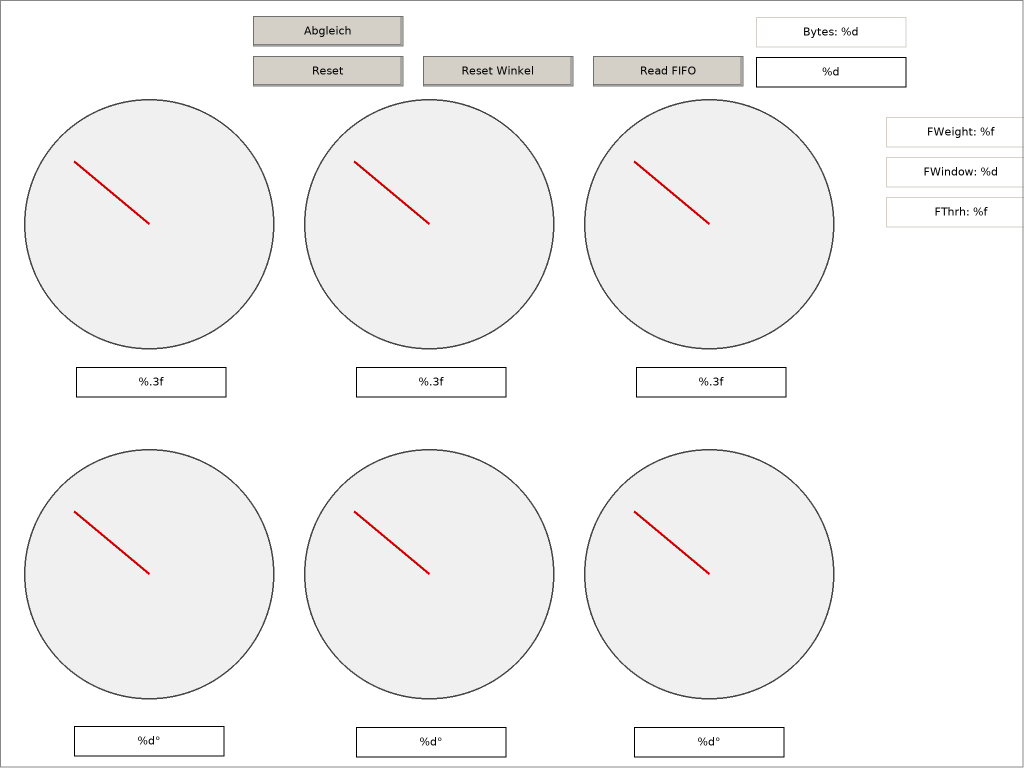
VISUALIZATION Visualization  // 1024x768
    Meter360 (24,99 250x250), value: MAIN.DegMovingHead[2], style: Meter-Meter360-Gray, scale format: %d, scale 0..360
    Rectangle (76,367 150x30), "%.3f", text variable: MAIN.Deg[0]
    Button (253,16 150x30), "Abgleich", colour toggle: MAIN.iFilter[0].bRingbufferFilled
        p2175578022: 16#ffffff
        p573394764: 16#FFFF8080
        tap MAIN.bWriteOffset
    Button (253,56 150x30), "Reset"
        tap MAIN.bReset
    Meter360 (304,99 250x250), value: MAIN.DegMovingHead[1], style: Meter-Meter360-Gray, scale format: %d, scale 0..360
    Rectangle (356,367 150x30), "%.3f", text variable: MAIN.Deg[1]
    Meter360 (584,99 250x250), value: MAIN.DegMovingHead[0], style: Meter-Meter360-Gray, scale format: %d, scale 0..360
    Rectangle (636,367 150x30), "%.3f", text variable: MAIN.Deg[0]
    Button (423,56 150x30), "Reset Winkel"
        tap MAIN.bResetAngle
    Button (593,56 150x30), "Read FIFO"
        tap MAIN.bReadFIFO
    Rectangle (756,57 150x30), "%d", text variable: MAIN.arBuf[2]
    Textfield (756,17 150x30), "Bytes: %d", text variable: MAIN.bytesToRead
        OnMouseClick: write the text variable via Default
    Meter360 (24,449 250x250), value: MAIN.degGamma, style: Meter-Meter360-Gray, scale format: %d, scale 0..360
    Meter360 (304,449 250x250), value: MAIN.degTheta, style: Meter-Meter360-Gray, scale format: %d, scale 0..360
    Meter360 (584,449 250x250), value: MAIN.degPhi, style: Meter-Meter360-Gray, scale format: %d, scale 0..360
    Textfield (886,117 150x30), "FWeight: %f", text variable: MAIN.fusionWeight
        OnMouseClick: write the text variable via Default
    Textfield (886,157 150x30), "FWindow: %d", text variable: MAIN.fusionWindow
        OnMouseClick: write the text variable via Default
    Textfield (886,197 150x30), "FThrh: %f", text variable: MAIN.fusionHorizontThreshold
        OnMouseClick: write the text variable via Default
    Rectangle (74,726 150x30), "%d°", text variable: MAIN.degGamma
    Rectangle (356,727 150x30), "%d°", text variable: MAIN.degTheta
    Rectangle (634,727 150x30), "%d°", text variable: MAIN.degTheta
END_VISUALIZATION

(* stored: Version 1.1.0.1, ProductVersion 3.1.4024.12
   Visu Visualization: Id {2bcdb9c8-65b9-4a3d-9749-96111609333d} *)
